// TIA Portal V18 export
// export: Created 2026-06-08T17:01:58.0830858Z, ExportSetting WithDefaults, DisplayName Totally Integrated Automation Portal, DisplayVersion V18, DisplayName TIA Portal Openness, DisplayVersion V18, DisplayName TIA Portal Version Control Interface, DisplayVersion V18, DisplayName STEP 7 Professional, DisplayVersion V18, DisplayName STEP 7 Safety, DisplayVersion V18, DisplayName WinCC Professional, DisplayVersion V18
DATA_BLOCK "STATES_DB"   // DB2
{ S7_Optimized_Access := 'FALSE' }
VERSION : 0.1
// stored: AutoNumber true, DBAccessibleFromOPCUA true, IsOnlyStoredInLoadMemory false, IsWriteProtectedInAS false
   VAR
      EMERGENCY_STATE : Bool;
      DIV_1 : Bool;
      DIV_2 : Bool;
      MAIN_WIND_DOWN : Bool;
      M1_WIND_DOWN : Bool;
      M2_WIND_DOWN : Bool;
      DIV1_COUNTING_READY : Bool;
      DIV2_COUNTING_READY : Bool;
   END_VAR
BEGIN
END_DATA_BLOCK
